Universal Robots PolyScope program: IAC001 PositionMove.urp

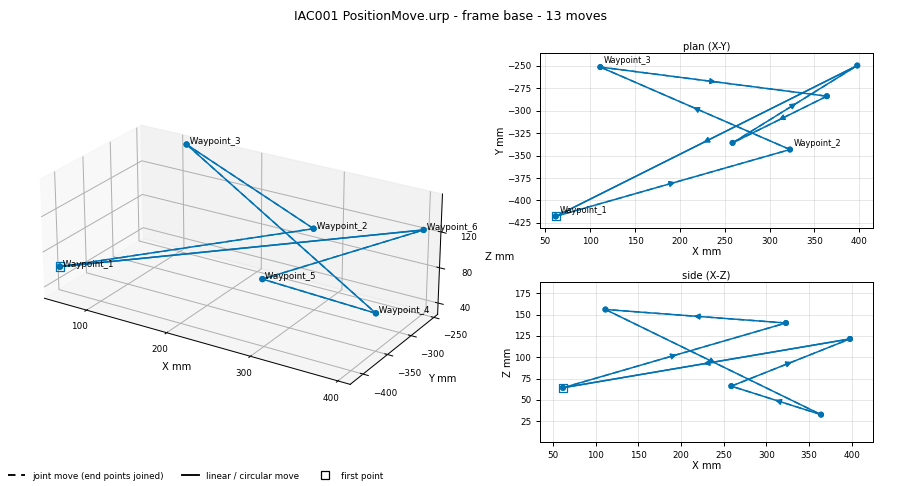
[picture p0: tool path of IAC001 PositionMove.urp in frame base, 13 of 13 moves have a stored position in this frame; points joined in program order, loops and branches not executed]
Program IAC001 PositionMove (installation=default directory=/programs createdIn=5.9.1.1031110 lastSavedIn=5.9.1.1031110 robotSerialNumber=20195501059)
Calibrated DH parameters: a=[0.000146, -0.418764, -0.053981, 0.000058, -0.000023, 0]; d=[0.162545, 37.319448, -206.067439, 168.881546, 0.09955, 0.099464]; alpha=[1.57004, -0.001979, 0.002304, 1.570607, -1.57066, 0]; deltaTheta=[0, -0.174616, -1.258233, 1.432844, -0.000001, 0]
Robot Program (runOnlyOnce=false)
  MoveJ speed 120 deg/s, acceleration 80 deg/s^2 (useActiveTCP=true positionType=JointAngles) feature=Base
    Waypoint Waypoint_1: TCP in base x=61.57 y=-417.708 z=64.277 mm, rx=0.8678 ry=3.0175 rz=-0.0002 rad; joints [79.864, -90.253, 129.777, -129.533, 270.177, 21.988] deg; TCP offset x=0 y=0 z=174 mm, rx=0 ry=0 rz=0 rad
    Waypoint Waypoint_2: TCP in base x=322.828 y=-343.188 z=140.145 mm, rx=0.8679 ry=3.0175 rz=-0.0002 rad; joints [116.727, -89.981, 116.31, -116.394, 270.12, 58.832] deg
    Waypoint Waypoint_3: TCP in base x=111.337 y=-251.239 z=155.96 mm, rx=0.8275 ry=2.8789 rz=-0.5235 rad; joints [81.201, -145.121, 149.252, -114.525, 273.297, 23.813] deg
    Waypoint Waypoint_4: TCP in base x=363.98 y=-283.703 z=32.774 mm, rx=-0.8479 ry=-2.9471 rz=-0.3212 rad; joints [121.176, -77.864, 119.323, -120.839, 276.526, 62.706] deg
    Waypoint Waypoint_5: TCP in base x=258.812 y=-335.755 z=66.164 mm, rx=1.6238 ry=2.1056 rz=-0.1964 rad; joints [101.539, -97.009, 152.135, -171.527, 281.223, 89.542] deg
    Waypoint Waypoint_6: TCP in base x=397.891 y=-249.499 z=121.504 mm, rx=-1.962 ry=-2.2466 rz=-0.7756 rad; joints [115.763, -85.845, 116.435, -104.938, 295.202, 104.518] deg
  MoveL speed 1000 mm/s, acceleration 1200 mm/s^2 (useActiveTCP=true) feature=Base
    Waypoint Waypoint_1: TCP in base x=61.57 y=-417.708 z=64.277 mm, rx=0.8678 ry=3.0175 rz=-0.0002 rad; joints [79.864, -90.253, 129.777, -129.533, 270.177, 21.988] deg
    Waypoint Waypoint_2: TCP in base x=322.828 y=-343.188 z=140.145 mm, rx=0.8679 ry=3.0175 rz=-0.0002 rad; joints [116.727, -89.981, 116.31, -116.394, 270.12, 58.832] deg
    Waypoint Waypoint_3: TCP in base x=111.337 y=-251.239 z=155.96 mm, rx=0.8275 ry=2.8789 rz=-0.5235 rad; joints [81.201, -145.121, 149.252, -114.525, 273.297, 23.813] deg
    Waypoint Waypoint_4: TCP in base x=363.98 y=-283.703 z=32.774 mm, rx=-0.8479 ry=-2.9471 rz=-0.3212 rad; joints [121.176, -77.864, 119.323, -120.839, 276.526, 62.706] deg
    Waypoint Waypoint_5: TCP in base x=258.812 y=-335.755 z=66.164 mm, rx=1.6238 ry=2.1056 rz=-0.1964 rad; joints [101.539, -97.009, 152.135, -171.527, 281.223, 89.542] deg
    Waypoint Waypoint_6: TCP in base x=397.891 y=-249.499 z=121.504 mm, rx=-1.962 ry=-2.2466 rz=-0.7756 rad; joints [115.763, -85.845, 116.435, -104.938, 295.202, 104.518] deg
  MoveL speed 250 mm/s, acceleration 1200 mm/s^2 (useActiveTCP=true) feature=Base
    Waypoint Waypoint_1: TCP in base x=61.57 y=-417.708 z=64.277 mm, rx=0.8678 ry=3.0175 rz=-0.0002 rad; joints [79.864, -90.253, 129.777, -129.533, 270.177, 21.988] deg
